// TIA Portal V16 export
// export: Created 2023-08-28T09:37:54.2707542Z, ExportSetting WithDefaults, DisplayName Totally Integrated Automation Portal, DisplayVersion V16 Update 6, DisplayName TIA Portal Version Control Interface, DisplayVersion V16 Update 2, DisplayName TIA Portal Openness, DisplayVersion V16 Update 6, DisplayName STEP 7 Professional, DisplayVersion V16 Update 6, DisplayName STEP 7 Safety, DisplayVersion V16, DisplayName WinCC Advanced, DisplayVersion V16 Update 6
VAR_GLOBAL   // PLC tag table "P2"
   inputReadyP2 AT %M82.1 : Bool;   // sugnał gotowość / Gotowość napędu
   inputRunF_P2 AT %M82.2 : Bool;   // stycznik falownik / Potwierdzenie pracy z falownika
   inputRunS_P2 AT %M82.3 : Bool;   // stycznik softstart / Powierdzenie pracy z sieci
   CMD_inverter_P2 AT %M82.4 : Bool;   // Stycznik Falownik
   CMD_network_P2 AT %M82.5 : Bool;   // Stycznik Sieć
   setCMD_FP2 AT %M207.2 : Bool;   // Znacznik sterowania w trybie falownik dlaP1
   setCMD_SP2 AT %M207.3 : Bool;   // Znacznik sterowania w trybie sieć
   IsReady_P2 AT %M17.1 : Bool;   // Znacznik gotowości napędu
   CB_CMD_P2 AT %M12.5 : Bool;   // Znacznik polecenia on/off przekaźnik napędu
   Set_HWork_P2 AT %M11.1 : Bool;   // Znacznik ustawienia aktywnej do pracy (po porównaniu liczników pracy)
   IsRunInverter_P2 AT %M211.4 : Bool;   // Potwierdzenie pracy z falownika
   IsRunNetwork_P2 AT %M217.1 : Bool;   // Potwierdzenie pracy z sieci
   Is_extras_K1_P2 AT %M218.5 : Bool;   // Znacznik motor dodatkowy nr 1
   setSUPV_FP2 AT %M12.1 : Bool;   // Znacznik polecenia startu z falownika
   IsRun_P2 AT %M10.5 : Bool;   // Potwierdzenie pracy
   setSUPV_SP2 AT %M13.0 : Bool;   // Znacznik polecenia startu z sieci
   CMD_soft_P2 AT %M85.0 : Bool;   // sygnał z softstart potwierdzenie pracy / sygnał on/off soft-start
   resetFault_SoftStart_P2 AT %M50.1 : Bool;   // sygnał resetu softstart
   bitH_Alarm_P2 AT %M62.0 : Bool;   // Alarm - kopia bitu z instancji statusu napędu
   bitH_REM_P2 AT %M62.2 : Bool;   // Zdalna - kopia bitu z instancji statusu napędu
   bitH_RUN_P2 AT %M62.3 : Bool;   // Praca - kopia bitu z instancji statusu napędu
   bitH_OFF_P2 AT %M62.4 : Bool;   // Polecenie OFF - kopia bitu z instancji statusu napędu
   bitH_ON_P2 AT %M62.5 : Bool;   // Polecenie ON - kopia bitu z instancji statusu napędu
   bitH_Res_P2 AT %M62.6 : Bool;   // Reset - kopia bitu z instancji statusu napędu
   bitH_Aut_Man_P2 AT %M62.7 : Bool;   // Aut=1 Man=0 - kopia bitu z instancji statusu napędu
   bitH_rezerwa_P2 AT %M62.1 : Bool;   // rez
   Is_extras_K3_P2 AT %M89.6 : Bool;   // Znacznik motor dodatkowy nr 3
   Is_extras_K2_P2 AT %M219.0 : Bool;   // Znacznik motor dodatkowy nr 2
   off_add_K1_P2 AT %M52.3 : Bool;   // sterowanie wyłączeniem selektywnym dodatkowej
   off_add_K2_P2 AT %M52.4 : Bool;   // sterowanie wyłączeniem selektywnym dodatkowej
   off_add_K3_P2 AT %M52.5 : Bool;   // sterowanie wyłączeniem selektywnym dodatkowej
   off_add_K4_P2 AT %M53.5 : Bool;   // sterowanie wyłączeniem selektywnym dodatkowej
   CMD_ErrorSet_NetworkP2 AT %M221.4 : Bool;   // Znacznik sterowania awaryjnego pracą pompy bez falownika
   Hour_Work_P2 AT %MD40 : DWord;   // Licznik pracy
   "Ustaw alarm P2" AT %M1040.3 : Bool;   // symulacyjny bit alarmu
   Set_50Hz_P2 AT %M217.7 : Bool;   // Znacznik pamięci podtrzymujący przełączenie na sieć
   Mem_Res_setCMD_MC_P2 AT %M223.1 : Bool;   // pamięć zbocza załączenia timera blokowania stycznika falowni
END_VAR
